FUNCTION_BLOCK FB_StationDerived EXTENDS FB_Station
VAR
	_nCycles	: UDINT;
END_VAR

Cyclic();

METHOD Cyclic
VAR
END_VAR
SUPER^.Cyclic();
_nCycles := _nCycles + 1;
END_METHOD

END_FUNCTION_BLOCK

(* stored: Version 1.1.0.1, ProductVersion 3.1.4024.12
   POU FB_StationDerived: Id {422bf86d-f1ab-4f87-bbf0-86131e211494}, SpecialFunc None
   Method Cyclic: Id {e30c34e9-e1d4-4431-939a-4aa6099d30a5} *)
